(* Logix 5000 project; controller BreakGroup_US vendor 1 type 14 code 211 rev 32.16; software revision 32.05; part 4 of 8 *)
(* tags used below, declared in another part *)
   Gantry_01Vertical_Limit_Switch_1 : ALIAS FOR MCP_PT01:23:I.0;
   Gantry_01Vertical_Limit_Switch_2 : ALIAS FOR MCP_PT01:23:I.1;
   Gantry_02_Vertical_Limit_Switch_1 : ALIAS FOR RCP_PT01:22:I.7;
   Gantry_02_Vertical_Limit_Switch_2 : ALIAS FOR RCP_PT01:23:I.0;
   Gantry_1_Clamping_Start_PB : ALIAS FOR MCP_PT01:24:I.5;
   Gantry_1_Clamping_Stop_PB : ALIAS FOR MCP_PT01:24:I.6;
   Gantry_1_EMG_PB : ALIAS FOR MCP_PT01:24:I.0;
   Gantry_1_Home_PB : ALIAS FOR MCP_PT01:24:I.7;
   Gantry_1_Horizontal_Limit_Switch_01 : ALIAS FOR MCP_PT01:22:I.4;
   Gantry_1_Horizontal_Limit_Switch_02 : ALIAS FOR MCP_PT01:22:I.5;
   Gantry_1_Horizontal_Start_PB : ALIAS FOR MCP_PT01:24:I.1;
   Gantry_1_Horizontal_Stop_PB : ALIAS FOR MCP_PT01:24:I.2;
   Gantry_1_LH_Clamping_Limit_Switch_1 : ALIAS FOR MCP_PT01:23:I.2;
   Gantry_1_LH_Clamping_Limit_Switch_2 : ALIAS FOR MCP_PT01:23:I.3;
   Gantry_1_RH_Clamping_Limit_Switch_1 : ALIAS FOR MCP_PT01:23:I.4;
   Gantry_1_RH_Clamping_Limit_Switch_2 : ALIAS FOR MCP_PT01:23:I.5;
   Gantry_1_Vertical_Locking_Cyl_1Extended : ALIAS FOR MCP_PT01:23:I.6;
   Gantry_1_Vertical_Locking_Cyl_1Retracted : ALIAS FOR MCP_PT01:23:I.7;
   Gantry_1_Vertical_Start_PB : ALIAS FOR MCP_PT01:24:I.3;
   Gantry_1_Vertical_Stop_PB : ALIAS FOR MCP_PT01:24:I.4;
   Gantry_1Collision_sensor : ALIAS FOR MCP_PT01:22:I.6;
   Gantry_1Zero_Pos_Sensor : ALIAS FOR MCP_PT01:22:I.7;
   Gantry_2_Clamping_Start_PB : ALIAS FOR RCP_PT01:24:I.6;
   Gantry_2_Clamping_Stop_PB : ALIAS FOR RCP_PT01:24:I.7;
   Gantry_2_Collision_sensor : ALIAS FOR RCP_PT01:22:I.5;
   Gantry_2_Emg_PB : ALIAS FOR RCP_PT01:24:I.1;
   Gantry_2_Horizontal_Limit_Switch_01 : ALIAS FOR RCP_PT01:22:I.3;
   Gantry_2_Horizontal_Limit_Switch_02 : ALIAS FOR RCP_PT01:22:I.4;
   Gantry_2_Horizontal_Start_PB : ALIAS FOR RCP_PT01:24:I.2;
   Gantry_2_Horizontal_Stop_PB : ALIAS FOR RCP_PT01:24:I.3;
   Gantry_2_LH_Clamping_Limit_Switch_1 : ALIAS FOR RCP_PT01:23:I.1;
   Gantry_2_LH_Clamping_Limit_Switch_2 : ALIAS FOR RCP_PT01:23:I.2;
   Gantry_2_LH_Tilting_Home_PositionSensor : ALIAS FOR RCP_PT01:23:I.7;
   Gantry_2_RH_Clamping_Limit_Switch_1 : ALIAS FOR RCP_PT01:23:I.3;
   Gantry_2_RH_Clamping_Limit_Switch_2 : ALIAS FOR RCP_PT01:23:I.4;
   Gantry_2_RH_Tilting_Home_PositionSensor : ALIAS FOR RCP_PT01:24:I.0;
   Gantry_2_Vertical_Locking_Cyl_1Extended : ALIAS FOR RCP_PT01:23:I.5;
   Gantry_2_Vertical_Locking_Cyl_1Retracted : ALIAS FOR RCP_PT01:23:I.6;
   Gantry_2_Vertical_Start_PB : ALIAS FOR RCP_PT01:24:I.4;
   Gantry_2_Vertical_Stop_PB : ALIAS FOR RCP_PT01:24:I.5;
   Gantry_2_Zero_Pos_Sensor : ALIAS FOR RCP_PT01:22:I.6;
   Out_ST30_Home_PB : ALIAS FOR MCP_PT01:26:O.7;
   Out_ST30_Hydro_Motor_On : ALIAS FOR MCP_PT01:26:O.4;
   Out_ST30_Index_PlateLockCyl1_Extend : ALIAS FOR MCP_PT01:25:O.4;
   Out_ST30_Index_PlateLockCyl1_Retract : ALIAS FOR MCP_PT01:25:O.5;
   Out_ST30_Index_PlateLockCyl2_Extend : ALIAS FOR MCP_PT01:25:O.6;
   Out_ST30_Index_PlateLockCyl2_Retract : ALIAS FOR MCP_PT01:25:O.7;
   Out_ST30_Press_Unit_Cyl_1Extend : ALIAS FOR MCP_PT01:26:O.0;
   Out_ST30_Press_Unit_Cyl_1Retract : ALIAS FOR MCP_PT01:26:O.1;
   Out_ST30_Press_Unit_Cyl_2Extend : ALIAS FOR MCP_PT01:26:O.2;
   Out_ST30_Press_Unit_Cyl_2Retract : ALIAS FOR MCP_PT01:26:O.3;
   Out_ST30_Reset_PB : ALIAS FOR MCP_PT01:27:O.0;
   Out_ST30_Servo_Healthy_Indication : ALIAS FOR MCP_PT01:27:O.1;
   Out_ST30_Servo_Trip_Indication : ALIAS FOR MCP_PT01:27:O.2;
   Out_ST30_Start_PB : ALIAS FOR MCP_PT01:26:O.5;
   Out_ST30_Stop_PB : ALIAS FOR MCP_PT01:26:O.6;
   Out_ST40_Home_PB : ALIAS FOR MCP_PT01:30:O.6;
   Out_ST40_Index_PlateLockCyl1_Extend : ALIAS FOR MCP_PT01:27:O.3;
   Out_ST40_Index_PlateLockCyl1_Retract : ALIAS FOR MCP_PT01:27:O.4;
   Out_ST40_Index_PlateLockCyl2_Extend : ALIAS FOR MCP_PT01:27:O.5;
   Out_ST40_Index_PlateLockCyl2_Retract : ALIAS FOR MCP_PT01:27:O.6;
   Out_ST40_Reset_PB : ALIAS FOR MCP_PT01:30:O.7;
   Out_ST40_Servo_Healthy_Indication : ALIAS FOR MCP_PT01:31:O.0;
   Out_ST40_Servo_Trip_Indication : ALIAS FOR MCP_PT01:31:O.1;
   Out_ST40_Start_PB : ALIAS FOR MCP_PT01:30:O.4;
   Out_ST40_Stop_PB : ALIAS FOR MCP_PT01:30:O.5;
   Out_ST_10_Trolley_1LockCylExtend : ALIAS FOR MCP_PT01:25:O.0;
   Out_ST_10_Trolley_1LockCylRetract : ALIAS FOR MCP_PT01:25:O.1;
   Out_ST_20_Trolley_1LockCylExtend : ALIAS FOR MCP_PT01:25:O.2;
   Out_ST_20_Trolley_1LockCylRetract : ALIAS FOR MCP_PT01:25:O.3;
   ST100_Auto_SS : ALIAS FOR RCP_PT01:14:I.3;
   ST100_Conv_End_Sensor : ALIAS FOR RCP_PT01:10:I.7;
   ST100_Conv_Home_Sensor : ALIAS FOR RCP_PT01:10:I.6;
   ST100_EMG_PB : ALIAS FOR RCP_PT01:13:I.5;
   ST100_Home_PB : ALIAS FOR RCP_PT01:14:I.2;
   ST100_IndexPlateLockCyl01_Extended : ALIAS FOR RCP_PT01:10:I.2;
   ST100_IndexPlateLockCyl01_Retracted : ALIAS FOR RCP_PT01:10:I.3;
   ST100_IndexPlateLockCyl02_Extended : ALIAS FOR RCP_PT01:10:I.4;
   ST100_IndexPlateLockCyl02_Retracted : ALIAS FOR RCP_PT01:10:I.5;
   ST100_IndexTableHomePositionSensor : ALIAS FOR RCP_PT01:10:I.1;
   ST100_Manual_SS : ALIAS FOR RCP_PT01:14:I.4;
   ST100_Product_Present_Sensor : ALIAS FOR RCP_PT01:10:I.0;
   ST100_Reset_PB : ALIAS FOR RCP_PT01:14:I.5;
   ST100_Start_1_PB : ALIAS FOR RCP_PT01:13:I.6;
   ST100_Start_2_PB : ALIAS FOR RCP_PT01:14:I.0;
   ST100_Stop_1_PB : ALIAS FOR RCP_PT01:13:I.7;
   ST100_Stop_2_PB : ALIAS FOR RCP_PT01:14:I.1;
   ST110_Auto_SS : ALIAS FOR RCP_PT01:17:I.2;
   ST110_Conv_End_Sensor : ALIAS FOR RCP_PT01:15:I.5;
   ST110_Conv_Home_Sensor : ALIAS FOR RCP_PT01:15:I.4;
   ST110_EMG_PB : ALIAS FOR RCP_PT01:16:I.4;
   ST110_Home_PB : ALIAS FOR RCP_PT01:17:I.1;
   ST110_IndexPlateLockCyl01_Extended : ALIAS FOR RCP_PT01:15:I.0;
   ST110_IndexPlateLockCyl01_Retracted : ALIAS FOR RCP_PT01:15:I.1;
   ST110_IndexPlateLockCyl02_Extended : ALIAS FOR RCP_PT01:15:I.2;
   ST110_IndexPlateLockCyl02_Retracted : ALIAS FOR RCP_PT01:15:I.3;
   ST110_IndexTableHomePositionSensor : ALIAS FOR RCP_PT01:14:I.7;
   ST110_Manual_SS : ALIAS FOR RCP_PT01:17:I.3;
   ST110_Product_Present_Sensor : ALIAS FOR RCP_PT01:14:I.6;
   ST110_Reset_PB : ALIAS FOR RCP_PT01:17:I.4;
   ST110_Start_1_PB : ALIAS FOR RCP_PT01:16:I.5;
   ST110_Start_2_PB : ALIAS FOR RCP_PT01:16:I.7;
   ST110_Stop_1_PB : ALIAS FOR RCP_PT01:16:I.6;
   ST110_Stop_2_PB : ALIAS FOR RCP_PT01:17:I.0;
   ST120_Auto_SS : ALIAS FOR RCP_PT01:22:I.0;
   ST120_Conv_End_Sensor : ALIAS FOR RCP_PT01:18:I.4;
   ST120_Conv_Home_Sensor : ALIAS FOR RCP_PT01:18:I.3;
   ST120_EMG_PB : ALIAS FOR RCP_PT01:21:I.2;
   ST120_Home_PB : ALIAS FOR RCP_PT01:21:I.7;
   ST120_IndexPlateLockCyl01_Extended : ALIAS FOR RCP_PT01:17:I.7;
   ST120_IndexPlateLockCyl01_Retracted : ALIAS FOR RCP_PT01:18:I.0;
   ST120_IndexPlateLockCyl02_Extended : ALIAS FOR RCP_PT01:18:I.1;
   ST120_IndexPlateLockCyl02_Retracted : ALIAS FOR RCP_PT01:18:I.2;
   ST120_IndexTableHomePositionSensor : ALIAS FOR RCP_PT01:17:I.6;
   ST120_Manual_SS : ALIAS FOR RCP_PT01:22:I.1;
   ST120_Product_Present_Sensor : ALIAS FOR RCP_PT01:17:I.5;
   ST120_Reset_PB : ALIAS FOR RCP_PT01:22:I.2;
   ST120_Start_1_PB : ALIAS FOR RCP_PT01:21:I.3;
   ST120_Start_2_PB : ALIAS FOR RCP_PT01:21:I.5;
   ST120_Stop_1_PB : ALIAS FOR RCP_PT01:21:I.4;
   ST120_Stop_2_PB : ALIAS FOR RCP_PT01:21:I.6;
   ST80_Auto_SS : ALIAS FOR RCP_PT01:6:I.0;
   ST80_Conv_End_Sensor : ALIAS FOR RCP_PT01:1:I.7;
   ST80_Conv_Home_Sensor : ALIAS FOR RCP_PT01:1:I.6;
   ST80_EMG_PB : ALIAS FOR RCP_PT01:5:I.2;
   ST80_Home_PB : ALIAS FOR RCP_PT01:5:I.7;
   ST80_Hydro_Motor : ALIAS FOR RCP_PT01:2:I.4;
   ST80_IndexPlateLockCyl01_Extended : ALIAS FOR RCP_PT01:1:I.2;
   ST80_IndexPlateLockCyl01_Retracted : ALIAS FOR RCP_PT01:1:I.3;
   ST80_IndexPlateLockCyl02_Extended : ALIAS FOR RCP_PT01:1:I.4;
   ST80_IndexPlateLockCyl02_Retracted : ALIAS FOR RCP_PT01:1:I.5;
   ST80_IndexTableHomePositionSensor : ALIAS FOR RCP_PT01:1:I.1;
   ST80_Manual_SS : ALIAS FOR RCP_PT01:6:I.1;
   ST80_Press_Unit_Cyl01_Extended : ALIAS FOR RCP_PT01:2:I.0;
   ST80_Press_Unit_Cyl01_Retracted : ALIAS FOR RCP_PT01:2:I.1;
   ST80_Press_Unit_Cyl02_Extended : ALIAS FOR RCP_PT01:2:I.2;
   ST80_Press_Unit_Cyl02_Retracted : ALIAS FOR RCP_PT01:2:I.3;
   ST80_Product_Present_Sensor : ALIAS FOR RCP_PT01:1:I.0;
   ST80_Reset_PB : ALIAS FOR RCP_PT01:6:I.2;
   ST80_Start_2_PB : ALIAS FOR RCP_PT01:5:I.5;
   ST80_Stop_2_PB : ALIAS FOR RCP_PT01:5:I.6;
   ST90_Auto_SS : ALIAS FOR RCP_PT01:9:I.5;
   ST90_Conv_End_Sensor : ALIAS FOR RCP_PT01:7:I.2;
   ST90_Conv_Home_Sensor : ALIAS FOR RCP_PT01:7:I.1;
   ST90_EMG_PB : ALIAS FOR RCP_PT01:8:I.7;
   ST90_Home_PB : ALIAS FOR RCP_PT01:9:I.4;
   ST90_IndexPlateLockCyl01_Extended : ALIAS FOR RCP_PT01:6:I.5;
   ST90_IndexPlateLockCyl01_Retracted : ALIAS FOR RCP_PT01:6:I.6;
   ST90_IndexPlateLockCyl02_Extended : ALIAS FOR RCP_PT01:6:I.7;
   ST90_IndexPlateLockCyl02_Retracted : ALIAS FOR RCP_PT01:7:I.0;
   ST90_IndexTableHomePositionSensor : ALIAS FOR RCP_PT01:6:I.4;
   ST90_Manual_SS : ALIAS FOR RCP_PT01:9:I.6;
   ST90_Product_Present_Sensor : ALIAS FOR RCP_PT01:6:I.3;
   ST90_Reset_PB : ALIAS FOR RCP_PT01:9:I.7;
   ST90_Start_1_PB : ALIAS FOR RCP_PT01:9:I.0;
   ST90_Start_2_PB : ALIAS FOR RCP_PT01:9:I.2;
   ST90_Stop_1_PB : ALIAS FOR RCP_PT01:9:I.1;
   ST90_Stop_2_PB : ALIAS FOR RCP_PT01:9:I.3;
(* MainProgram, continued *)

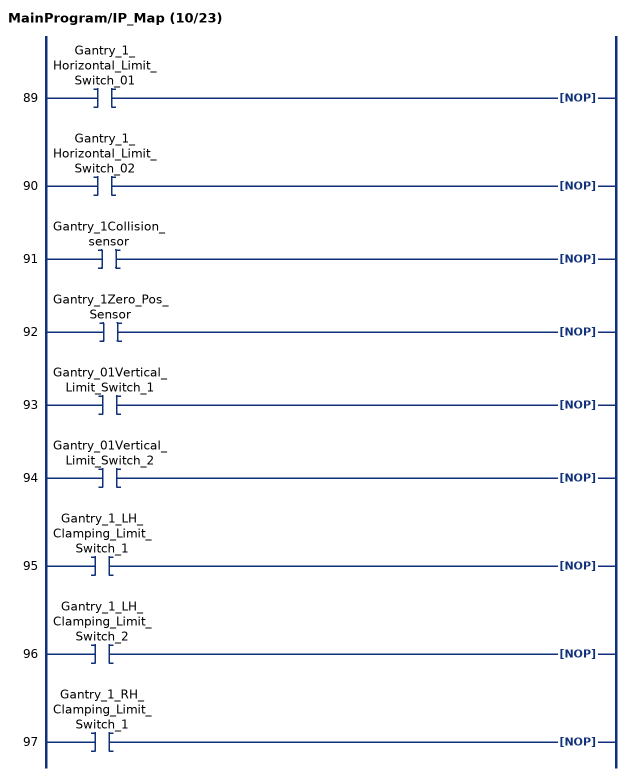
   89: XIC(Gantry_1_Horizontal_Limit_Switch_01)NOP();
   90: XIC(Gantry_1_Horizontal_Limit_Switch_02)NOP();
   91: XIC(Gantry_1Collision_sensor)NOP();
   92: XIC(Gantry_1Zero_Pos_Sensor)NOP();
   93: XIC(Gantry_01Vertical_Limit_Switch_1)NOP();
   94: XIC(Gantry_01Vertical_Limit_Switch_2)NOP();
   95: XIC(Gantry_1_LH_Clamping_Limit_Switch_1)NOP();
   96: XIC(Gantry_1_LH_Clamping_Limit_Switch_2)NOP();
   97: XIC(Gantry_1_RH_Clamping_Limit_Switch_1)NOP();
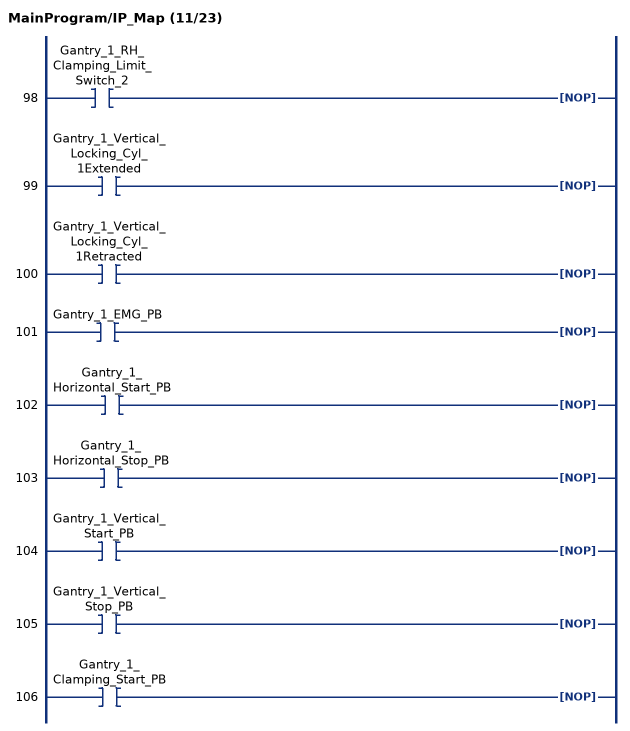
   98: XIC(Gantry_1_RH_Clamping_Limit_Switch_2)NOP();
   99: XIC(Gantry_1_Vertical_Locking_Cyl_1Extended)NOP();
   100: XIC(Gantry_1_Vertical_Locking_Cyl_1Retracted)NOP();
   101: XIC(Gantry_1_EMG_PB)NOP();
   102: XIC(Gantry_1_Horizontal_Start_PB)NOP();
   103: XIC(Gantry_1_Horizontal_Stop_PB)NOP();
   104: XIC(Gantry_1_Vertical_Start_PB)NOP();
   105: XIC(Gantry_1_Vertical_Stop_PB)NOP();
   106: XIC(Gantry_1_Clamping_Start_PB)NOP();
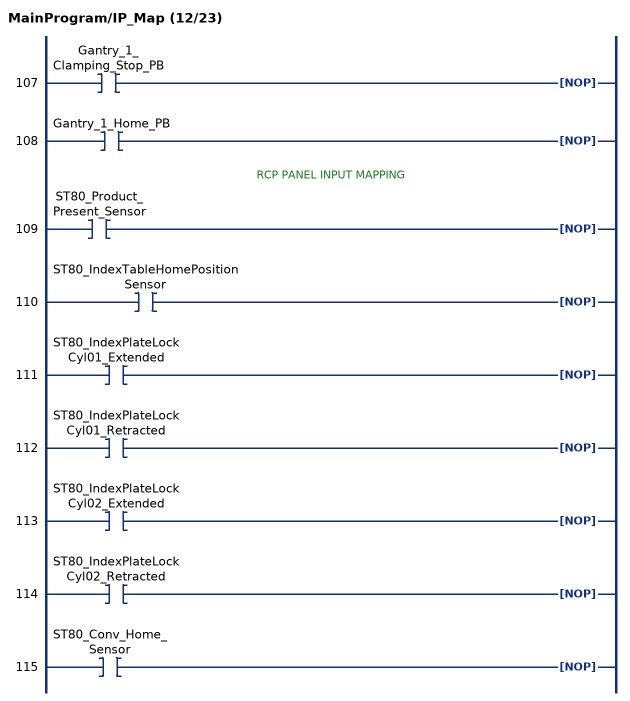
   107: XIC(Gantry_1_Clamping_Stop_PB)NOP();
   108: XIC(Gantry_1_Home_PB)NOP();
   // RCP PANEL INPUT MAPPING
   109: XIC(ST80_Product_Present_Sensor)NOP();
   110: XIC(ST80_IndexTableHomePositionSensor)NOP();
   111: XIC(ST80_IndexPlateLockCyl01_Extended)NOP();
   112: XIC(ST80_IndexPlateLockCyl01_Retracted)NOP();
   113: XIC(ST80_IndexPlateLockCyl02_Extended)NOP();
   114: XIC(ST80_IndexPlateLockCyl02_Retracted)NOP();
   115: XIC(ST80_Conv_Home_Sensor)NOP();
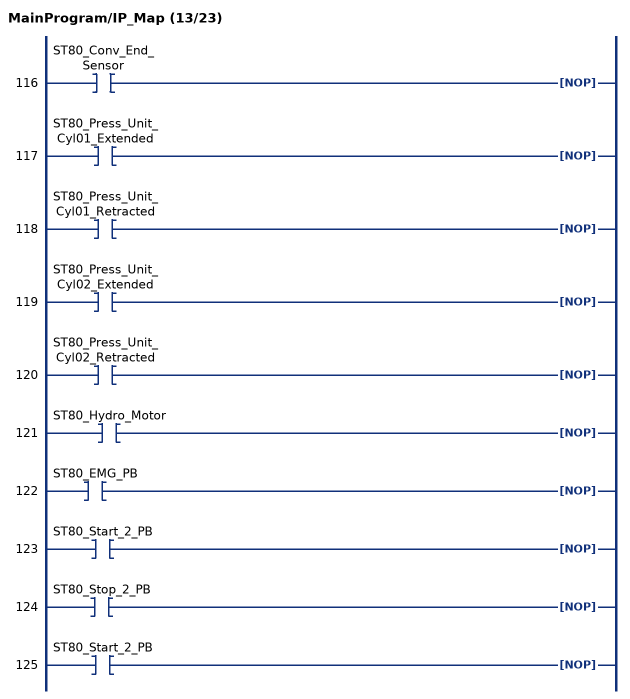
   116: XIC(ST80_Conv_End_Sensor)NOP();
   117: XIC(ST80_Press_Unit_Cyl01_Extended)NOP();
   118: XIC(ST80_Press_Unit_Cyl01_Retracted)NOP();
   119: XIC(ST80_Press_Unit_Cyl02_Extended)NOP();
   120: XIC(ST80_Press_Unit_Cyl02_Retracted)NOP();
   121: XIC(ST80_Hydro_Motor)NOP();
   122: XIC(ST80_EMG_PB)NOP();
   123: XIC(ST80_Start_2_PB)NOP();
   124: XIC(ST80_Stop_2_PB)NOP();
   125: XIC(ST80_Start_2_PB)NOP();
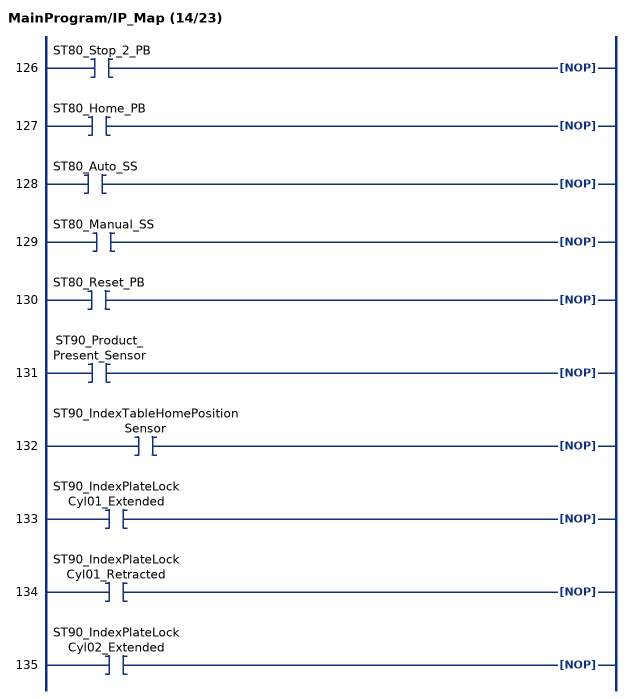
   126: XIC(ST80_Stop_2_PB)NOP();
   127: XIC(ST80_Home_PB)NOP();
   128: XIC(ST80_Auto_SS)NOP();
   129: XIC(ST80_Manual_SS)NOP();
   130: XIC(ST80_Reset_PB)NOP();
   131: XIC(ST90_Product_Present_Sensor)NOP();
   132: XIC(ST90_IndexTableHomePositionSensor)NOP();
   133: XIC(ST90_IndexPlateLockCyl01_Extended)NOP();
   134: XIC(ST90_IndexPlateLockCyl01_Retracted)NOP();
   135: XIC(ST90_IndexPlateLockCyl02_Extended)NOP();
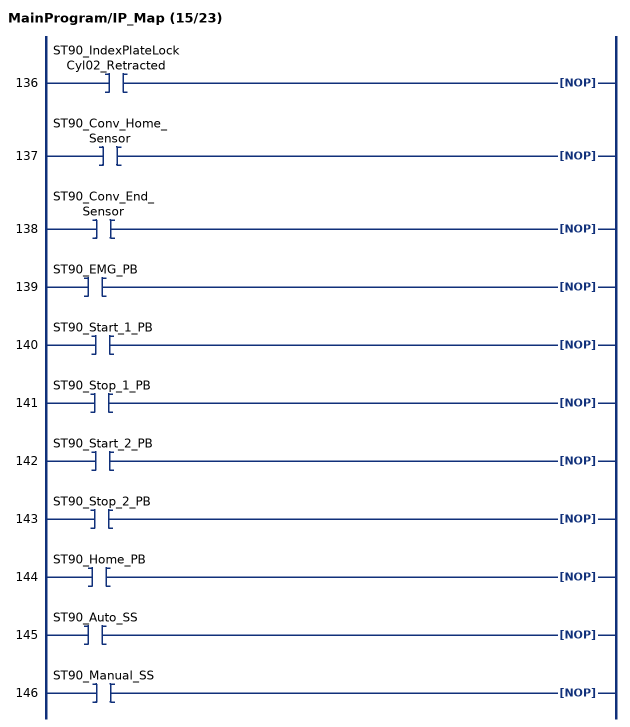
   136: XIC(ST90_IndexPlateLockCyl02_Retracted)NOP();
   137: XIC(ST90_Conv_Home_Sensor)NOP();
   138: XIC(ST90_Conv_End_Sensor)NOP();
   139: XIC(ST90_EMG_PB)NOP();
   140: XIC(ST90_Start_1_PB)NOP();
   141: XIC(ST90_Stop_1_PB)NOP();
   142: XIC(ST90_Start_2_PB)NOP();
   143: XIC(ST90_Stop_2_PB)NOP();
   144: XIC(ST90_Home_PB)NOP();
   145: XIC(ST90_Auto_SS)NOP();
   146: XIC(ST90_Manual_SS)NOP();
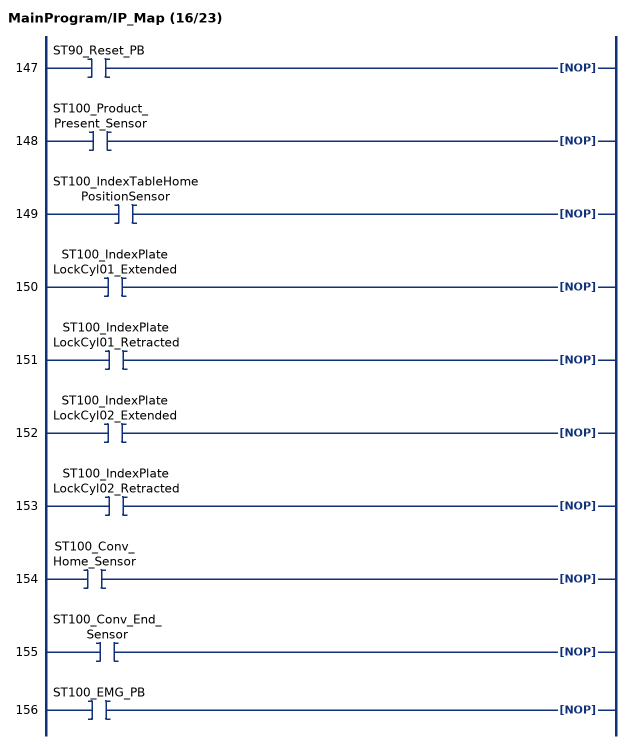
   147: XIC(ST90_Reset_PB)NOP();
   148: XIC(ST100_Product_Present_Sensor)NOP();
   149: XIC(ST100_IndexTableHomePositionSensor)NOP();
   150: XIC(ST100_IndexPlateLockCyl01_Extended)NOP();
   151: XIC(ST100_IndexPlateLockCyl01_Retracted)NOP();
   152: XIC(ST100_IndexPlateLockCyl02_Extended)NOP();
   153: XIC(ST100_IndexPlateLockCyl02_Retracted)NOP();
   154: XIC(ST100_Conv_Home_Sensor)NOP();
   155: XIC(ST100_Conv_End_Sensor)NOP();
   156: XIC(ST100_EMG_PB)NOP();
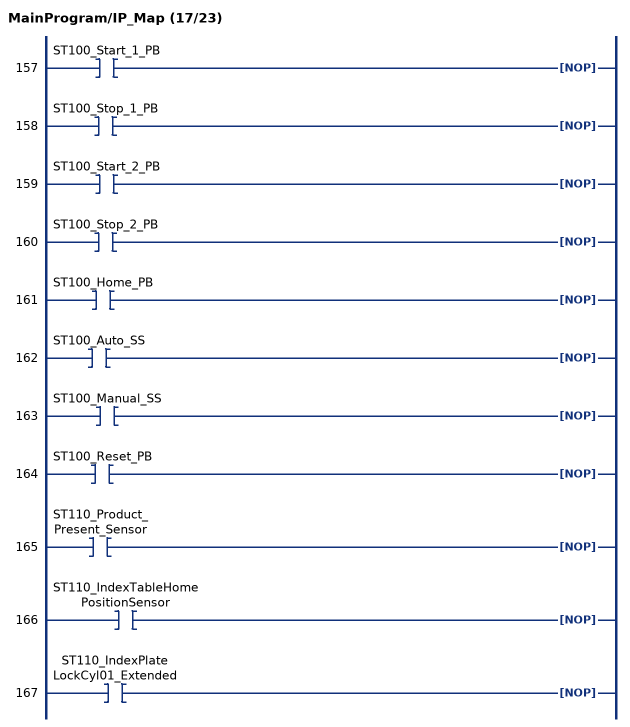
   157: XIC(ST100_Start_1_PB)NOP();
   158: XIC(ST100_Stop_1_PB)NOP();
   159: XIC(ST100_Start_2_PB)NOP();
   160: XIC(ST100_Stop_2_PB)NOP();
   161: XIC(ST100_Home_PB)NOP();
   162: XIC(ST100_Auto_SS)NOP();
   163: XIC(ST100_Manual_SS)NOP();
   164: XIC(ST100_Reset_PB)NOP();
   165: XIC(ST110_Product_Present_Sensor)NOP();
   166: XIC(ST110_IndexTableHomePositionSensor)NOP();
   167: XIC(ST110_IndexPlateLockCyl01_Extended)NOP();
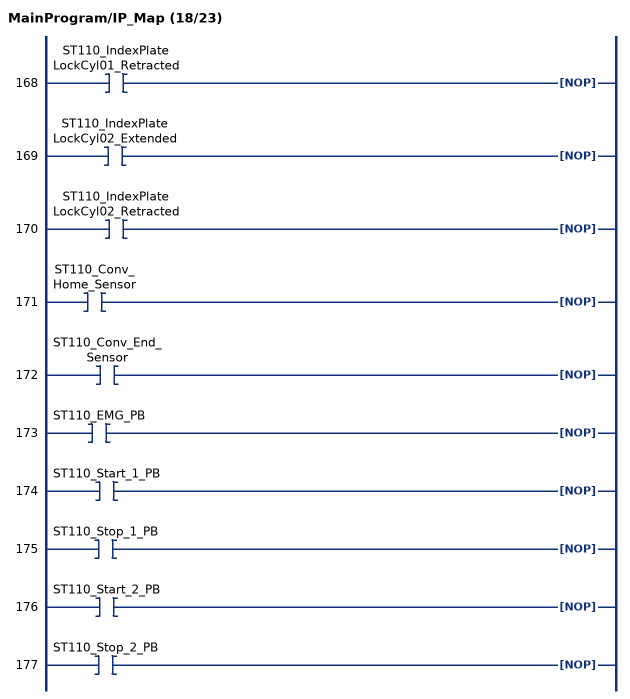
   168: XIC(ST110_IndexPlateLockCyl01_Retracted)NOP();
   169: XIC(ST110_IndexPlateLockCyl02_Extended)NOP();
   170: XIC(ST110_IndexPlateLockCyl02_Retracted)NOP();
   171: XIC(ST110_Conv_Home_Sensor)NOP();
   172: XIC(ST110_Conv_End_Sensor)NOP();
   173: XIC(ST110_EMG_PB)NOP();
   174: XIC(ST110_Start_1_PB)NOP();
   175: XIC(ST110_Stop_1_PB)NOP();
   176: XIC(ST110_Start_2_PB)NOP();
   177: XIC(ST110_Stop_2_PB)NOP();
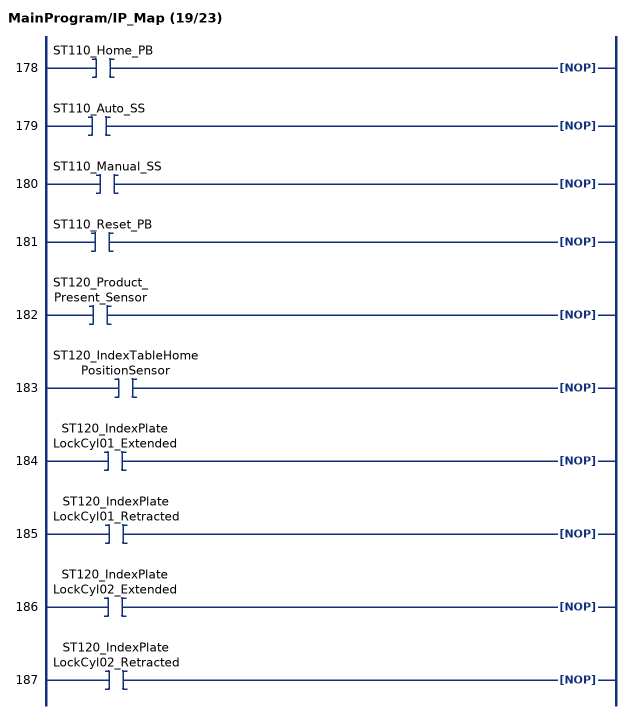
   178: XIC(ST110_Home_PB)NOP();
   179: XIC(ST110_Auto_SS)NOP();
   180: XIC(ST110_Manual_SS)NOP();
   181: XIC(ST110_Reset_PB)NOP();
   182: XIC(ST120_Product_Present_Sensor)NOP();
   183: XIC(ST120_IndexTableHomePositionSensor)NOP();
   184: XIC(ST120_IndexPlateLockCyl01_Extended)NOP();
   185: XIC(ST120_IndexPlateLockCyl01_Retracted)NOP();
   186: XIC(ST120_IndexPlateLockCyl02_Extended)NOP();
   187: XIC(ST120_IndexPlateLockCyl02_Retracted)NOP();
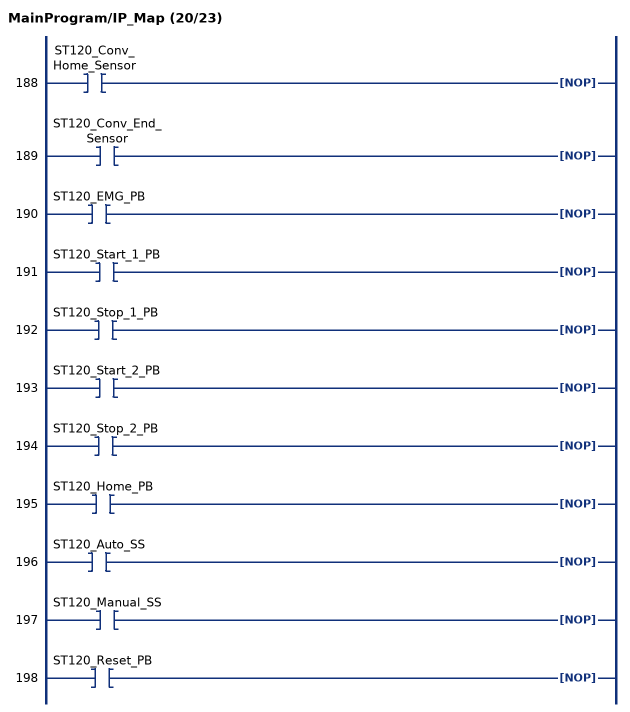
   188: XIC(ST120_Conv_Home_Sensor)NOP();
   189: XIC(ST120_Conv_End_Sensor)NOP();
   190: XIC(ST120_EMG_PB)NOP();
   191: XIC(ST120_Start_1_PB)NOP();
   192: XIC(ST120_Stop_1_PB)NOP();
   193: XIC(ST120_Start_2_PB)NOP();
   194: XIC(ST120_Stop_2_PB)NOP();
   195: XIC(ST120_Home_PB)NOP();
   196: XIC(ST120_Auto_SS)NOP();
   197: XIC(ST120_Manual_SS)NOP();
   198: XIC(ST120_Reset_PB)NOP();
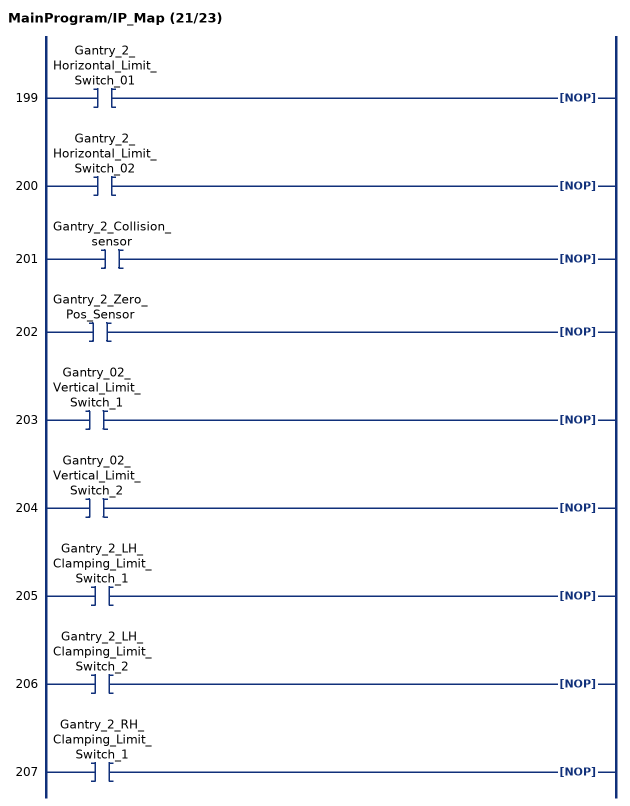
   199: XIC(Gantry_2_Horizontal_Limit_Switch_01)NOP();
   200: XIC(Gantry_2_Horizontal_Limit_Switch_02)NOP();
   201: XIC(Gantry_2_Collision_sensor)NOP();
   202: XIC(Gantry_2_Zero_Pos_Sensor)NOP();
   203: XIC(Gantry_02_Vertical_Limit_Switch_1)NOP();
   204: XIC(Gantry_02_Vertical_Limit_Switch_2)NOP();
   205: XIC(Gantry_2_LH_Clamping_Limit_Switch_1)NOP();
   206: XIC(Gantry_2_LH_Clamping_Limit_Switch_2)NOP();
   207: XIC(Gantry_2_RH_Clamping_Limit_Switch_1)NOP();
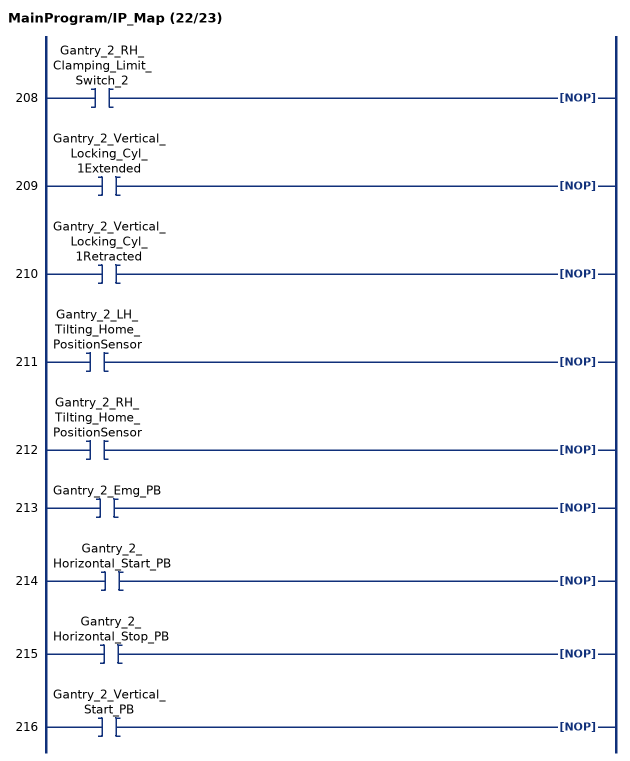
   208: XIC(Gantry_2_RH_Clamping_Limit_Switch_2)NOP();
   209: XIC(Gantry_2_Vertical_Locking_Cyl_1Extended)NOP();
   210: XIC(Gantry_2_Vertical_Locking_Cyl_1Retracted)NOP();
   211: XIC(Gantry_2_LH_Tilting_Home_PositionSensor)NOP();
   212: XIC(Gantry_2_RH_Tilting_Home_PositionSensor)NOP();
   213: XIC(Gantry_2_Emg_PB)NOP();
   214: XIC(Gantry_2_Horizontal_Start_PB)NOP();
   215: XIC(Gantry_2_Horizontal_Stop_PB)NOP();
   216: XIC(Gantry_2_Vertical_Start_PB)NOP();
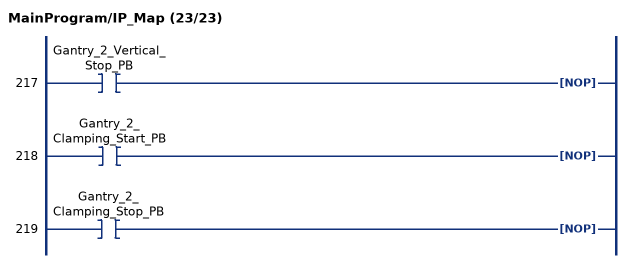
   217: XIC(Gantry_2_Vertical_Stop_PB)NOP();
   218: XIC(Gantry_2_Clamping_Start_PB)NOP();
   219: XIC(Gantry_2_Clamping_Stop_PB)NOP();
END_ROUTINE

ROUTINE Main   (* ladder *)
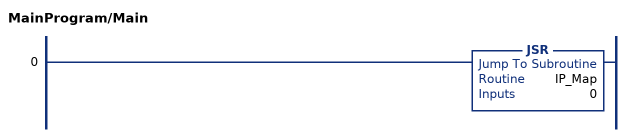
   0: JSR(IP_Map,0);
END_ROUTINE

ROUTINE OP_Map   (* ladder *)
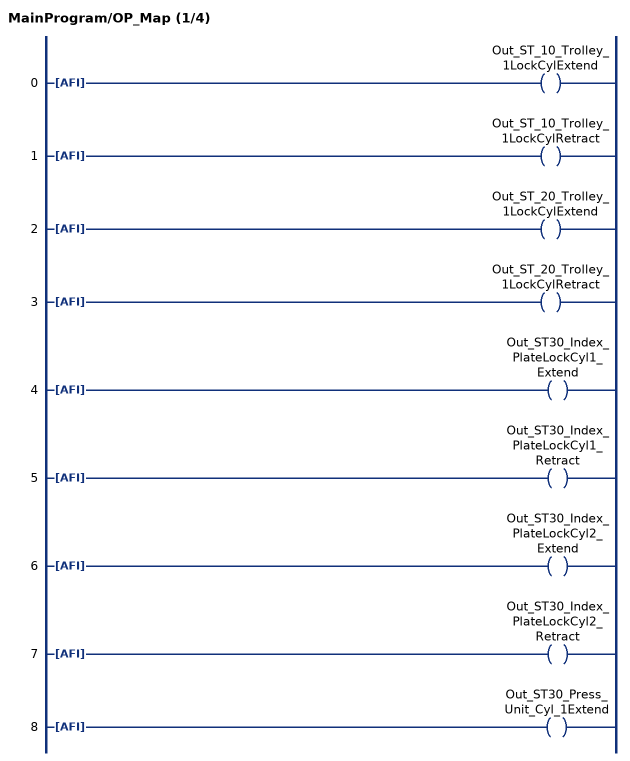
   0: AFI()OTE(Out_ST_10_Trolley_1LockCylExtend);
   1: AFI()OTE(Out_ST_10_Trolley_1LockCylRetract);
   2: AFI()OTE(Out_ST_20_Trolley_1LockCylExtend);
   3: AFI()OTE(Out_ST_20_Trolley_1LockCylRetract);
   4: AFI()OTE(Out_ST30_Index_PlateLockCyl1_Extend);
   5: AFI()OTE(Out_ST30_Index_PlateLockCyl1_Retract);
   6: AFI()OTE(Out_ST30_Index_PlateLockCyl2_Extend);
   7: AFI()OTE(Out_ST30_Index_PlateLockCyl2_Retract);
   8: AFI()OTE(Out_ST30_Press_Unit_Cyl_1Extend);
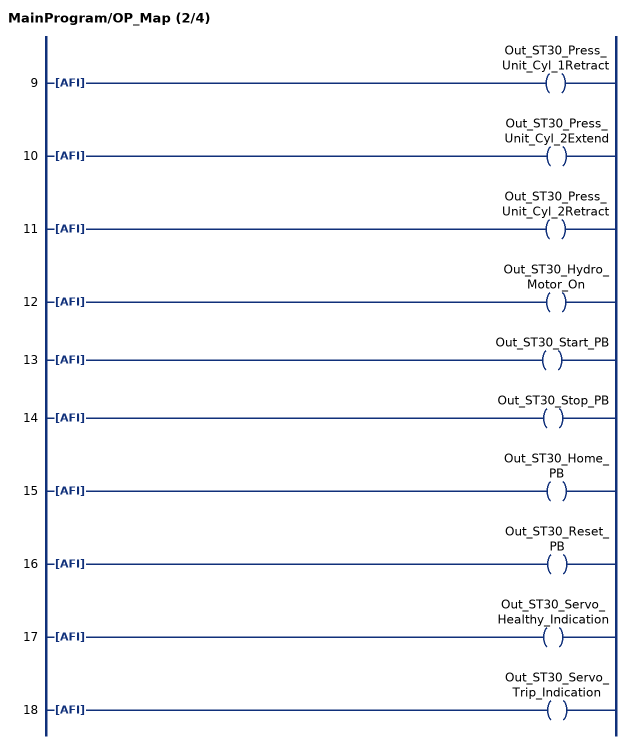
   9: AFI()OTE(Out_ST30_Press_Unit_Cyl_1Retract);
   10: AFI()OTE(Out_ST30_Press_Unit_Cyl_2Extend);
   11: AFI()OTE(Out_ST30_Press_Unit_Cyl_2Retract);
   12: AFI()OTE(Out_ST30_Hydro_Motor_On);
   13: AFI()OTE(Out_ST30_Start_PB);
   14: AFI()OTE(Out_ST30_Stop_PB);
   15: AFI()OTE(Out_ST30_Home_PB);
   16: AFI()OTE(Out_ST30_Reset_PB);
   17: AFI()OTE(Out_ST30_Servo_Healthy_Indication);
   18: AFI()OTE(Out_ST30_Servo_Trip_Indication);
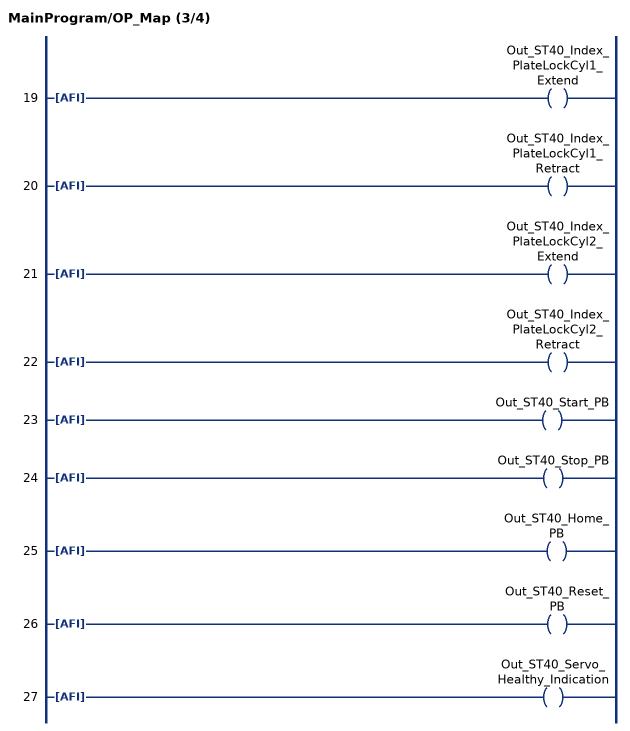
   19: AFI()OTE(Out_ST40_Index_PlateLockCyl1_Extend);
   20: AFI()OTE(Out_ST40_Index_PlateLockCyl1_Retract);
   21: AFI()OTE(Out_ST40_Index_PlateLockCyl2_Extend);
   22: AFI()OTE(Out_ST40_Index_PlateLockCyl2_Retract);
   23: AFI()OTE(Out_ST40_Start_PB);
   24: AFI()OTE(Out_ST40_Stop_PB);
   25: AFI()OTE(Out_ST40_Home_PB);
   26: AFI()OTE(Out_ST40_Reset_PB);
   27: AFI()OTE(Out_ST40_Servo_Healthy_Indication);
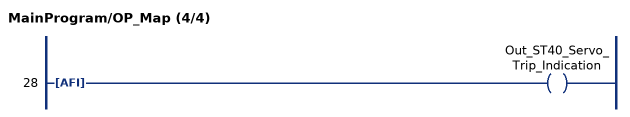
   28: AFI()OTE(Out_ST40_Servo_Trip_Indication);
END_ROUTINE
END_PROGRAM
